FUNCTION_BLOCK DigitalInput_HMI (* Service Interface Function Block Type *)
  (* Standard: 61499-2 *)
  (* Version 0.0, 6/15/2026, Schneider Electric, template *)
  PACKAGE SE.Nereda;
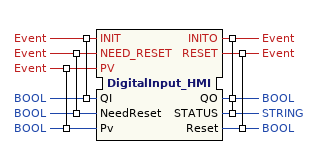
  EVENT_INPUT
    INIT WITH QI;
    NEED_RESET WITH NeedReset;
    PV WITH Pv;
  END_EVENT
  EVENT_OUTPUT
    INITO WITH QO, STATUS;
    RESET WITH Reset;
  END_EVENT
  VAR_INPUT
    QI : BOOL;
    NeedReset : BOOL;
    Pv : BOOL;
  END_VAR
  VAR_OUTPUT
    QO : BOOL; (* Event Output Qualifier *)
    STATUS : STRING; (* Service Status *)
    Reset : BOOL;
  END_VAR
  SERVICE /
    SEQUENCE 
    END_SEQUENCE
  END_SERVICE
END_FUNCTION_BLOCK
